// TIA Portal V16 export
// export: Created 2025-05-30T16:36:27.2401073Z, ExportSetting WithDefaults, DisplayName Totally Integrated Automation Portal, DisplayVersion V16, DisplayName TIA Portal Version Control Interface, DisplayVersion V16, DisplayName TIA Portal Openness, DisplayVersion V16, DisplayName STEP 7 Professional, DisplayVersion V16, DisplayName STEP 7 Safety, DisplayVersion V16, DisplayName WinCC Advanced, DisplayVersion V16
DATA_BLOCK "ProductBuffer_V3_DB"   // DB90
VERSION : 0.1
// stored: AutoNumber true, InstanceOfName ProductBuffer_V3, InstanceOfType FB
"ProductBuffer_V3"
   // VAR_INPUT
   //    SensorInput : Bool;
   //    EncoderPosition : Real;
   //    TriggerDistance : Real;
   //    TriggerFeedback : Bool;
   // END_VAR
   // VAR_OUTPUT
   //    TriggerMovement : Bool;
   //    ProductCount : Int;
   // END_VAR
   // VAR RETAIN
   //    ProductBuffer : Array[0..9] of "ProductTrack";
   //    PrevSensor { S7_SetPoint := 'True'} : Bool;
   //    MovementActive : Bool;
   //    i : Int;
   //    Distance : Real;
   // END_VAR
BEGIN
END_DATA_BLOCK
